// TIA Portal V20 export
DATA_BLOCK "DB_OPC_AnalogInputs"   // DB83
{ S7_Optimized_Access := 'TRUE' }
// stored: MemoryReserve 100
   VAR
      NumberOfSignals : Int := 22;
      Parameters : Struct
         Delay : LReal;
         DiffErrorMax : LReal;
         DiffErrorMin : LReal;
         DiffWarnMax : LReal;
         DiffWarnMin : LReal;
         Id : DInt;
         ItemNumber : DInt;
         Offset : LReal := 1.0;
         Gain : LReal;
         Target : LReal;
      END_STRUCT;
      Signals : Array[0..100] of "UDT_OPC_Analog";
      Update { S7_SetPoint := 'True'} : Bool;
   END_VAR
BEGIN
   // Signals[1].DiffErrorMax : Unit:W
   // Signals[3].DiffErrorMax : Unit:bar
   // Signals[4].DiffErrorMax : Unit:°C
   // Signals[5].DiffErrorMax : Unit:°C
   // Signals[6].DiffErrorMax : Unit:°C
   // Signals[7].DiffErrorMax : Unit:°C
   // Signals[8].DiffErrorMax : Unit:°C
   // Signals[9].DiffErrorMax : Unit:°C
   // Signals[10].DiffErrorMax : Unit:°C
   // Signals[13].DiffErrorMax : Unit:bar
   // Signals[14].DiffErrorMax : Unit:bar
   // Signals[15].DiffErrorMax : Unit:bar
   // Signals[16].DiffErrorMax : Unit:bar
   // Signals[17].DiffErrorMax : Unit:bar
   // Signals[18].DiffErrorMax : Unit:mm/s
   // Signals[19].DiffErrorMax : Unit:mm/s
   // Signals[21].DiffErrorMax : Unit:°C
   // Signals[26].DiffErrorMax : Unit:°C
   // Signals[1].DiffErrorMin : Unit:W
   // Signals[3].DiffErrorMin : Unit:bar
   // Signals[4].DiffErrorMin : Unit:°C
   // Signals[5].DiffErrorMin : Unit:°C
   // Signals[6].DiffErrorMin : Unit:°C
   // Signals[7].DiffErrorMin : Unit:°C
   // Signals[8].DiffErrorMin : Unit:°C
   // Signals[9].DiffErrorMin : Unit:°C
   // Signals[10].DiffErrorMin : Unit:°C
   // Signals[13].DiffErrorMin : Unit:bar
   // Signals[14].DiffErrorMin : Unit:bar
   // Signals[15].DiffErrorMin : Unit:bar
   // Signals[16].DiffErrorMin : Unit:bar
   // Signals[17].DiffErrorMin : Unit:bar
   // Signals[18].DiffErrorMin : Unit:mm/s
   // Signals[19].DiffErrorMin : Unit:mm/s
   // Signals[21].DiffErrorMin : Unit:°C
   // Signals[26].DiffErrorMin : Unit:°C
   // Signals[1].DiffWarnMax : Unit:W
   // Signals[3].DiffWarnMax : Unit:bar
   // Signals[4].DiffWarnMax : Unit:°C
   // Signals[5].DiffWarnMax : Unit:°C
   // Signals[6].DiffWarnMax : Unit:°C
   // Signals[7].DiffWarnMax : Unit:°C
   // Signals[8].DiffWarnMax : Unit:°C
   // Signals[9].DiffWarnMax : Unit:°C
   // Signals[10].DiffWarnMax : Unit:°C
   // Signals[13].DiffWarnMax : Unit:bar
   // Signals[14].DiffWarnMax : Unit:bar
   // Signals[15].DiffWarnMax : Unit:bar
   // Signals[16].DiffWarnMax : Unit:bar
   // Signals[17].DiffWarnMax : Unit:bar
   // Signals[18].DiffWarnMax : Unit:mm/s
   // Signals[19].DiffWarnMax : Unit:mm/s
   // Signals[21].DiffWarnMax : Unit:°C
   // Signals[26].DiffWarnMax : Unit:°C
   // Signals[1].DiffWarnMin : Unit:W
   // Signals[3].DiffWarnMin : Unit:bar
   // Signals[4].DiffWarnMin : Unit:°C
   // Signals[5].DiffWarnMin : Unit:°C
   // Signals[6].DiffWarnMin : Unit:°C
   // Signals[7].DiffWarnMin : Unit:°C
   // Signals[8].DiffWarnMin : Unit:°C
   // Signals[9].DiffWarnMin : Unit:°C
   // Signals[10].DiffWarnMin : Unit:°C
   // Signals[13].DiffWarnMin : Unit:bar
   // Signals[14].DiffWarnMin : Unit:bar
   // Signals[15].DiffWarnMin : Unit:bar
   // Signals[16].DiffWarnMin : Unit:bar
   // Signals[17].DiffWarnMin : Unit:bar
   // Signals[18].DiffWarnMin : Unit:mm/s
   // Signals[19].DiffWarnMin : Unit:mm/s
   // Signals[21].DiffWarnMin : Unit:°C
   // Signals[26].DiffWarnMin : Unit:°C
   // Signals[1].Offset : Unit:W
   // Signals[3].Offset : Unit:bar
   // Signals[4].Offset : Unit:°C
   // Signals[5].Offset : Unit:°C
   // Signals[6].Offset : Unit:°C
   // Signals[7].Offset : Unit:°C
   // Signals[8].Offset : Unit:°C
   // Signals[9].Offset : Unit:°C
   // Signals[10].Offset : Unit:°C
   // Signals[13].Offset : Unit:bar
   // Signals[14].Offset : Unit:bar
   // Signals[15].Offset : Unit:bar
   // Signals[16].Offset : Unit:bar
   // Signals[17].Offset : Unit:bar
   // Signals[18].Offset : Unit:mm/s
   // Signals[19].Offset : Unit:mm/s
   // Signals[21].Offset : Unit:°C
   // Signals[26].Offset : Unit:°C
   // Signals[1].Target : Unit:W
   // Signals[3].Target : Unit:bar
   // Signals[4].Target : Unit:°C
   // Signals[5].Target : Unit:°C
   // Signals[6].Target : Unit:°C
   // Signals[7].Target : Unit:°C
   // Signals[8].Target : Unit:°C
   // Signals[9].Target : Unit:°C
   // Signals[10].Target : Unit:°C
   // Signals[13].Target : Unit:bar
   // Signals[14].Target : Unit:bar
   // Signals[15].Target : Unit:bar
   // Signals[16].Target : Unit:bar
   // Signals[17].Target : Unit:bar
   // Signals[18].Target : Unit:mm/s
   // Signals[19].Target : Unit:mm/s
   // Signals[21].Target : Unit:°C
   // Signals[26].Target : Unit:°C
   // Signals[1].Value : Unit:W
   // Signals[3].Value : Unit:bar
   // Signals[4].Value : Unit:°C
   // Signals[5].Value : Unit:°C
   // Signals[6].Value : Unit:°C
   // Signals[7].Value : Unit:°C
   // Signals[8].Value : Unit:°C
   // Signals[9].Value : Unit:°C
   // Signals[10].Value : Unit:°C
   // Signals[13].Value : Unit:bar
   // Signals[14].Value : Unit:bar
   // Signals[15].Value : Unit:bar
   // Signals[16].Value : Unit:bar
   // Signals[17].Value : Unit:bar
   // Signals[18].Value : Unit:mm/s
   // Signals[19].Value : Unit:mm/s
   // Signals[21].Value : Unit:°C
   // Signals[26].Value : Unit:°C
END_DATA_BLOCK
